{attribute 'qualified_only'}
{attribute 'strict'}
TYPE States :
(
	GRIPPER_OPEN := 0,
	ROTATE_DISC := 1,
	LINEAR_FW := 2,
	GRIPPER_LOWER := 3,
	GRIPPER_CLOSE := 4,
	GRIPPER_LIFT := 5,
	LINEAR_BW := 6
);
END_TYPE

(* stored: Version 1.1.0.1, ProductVersion 3.1.4024.12
   DUT States: Id {40a30a0e-e35a-4d83-907a-269356be2a3a} *)
